TYPE DUT_HMI_General :
STRUCT
	Manuals 	: DUT_HMI_General_Manuals;		// Fanuc 
	Mes			: DUT_HMI_MesManual;
END_STRUCT
END_TYPE

(* stored: Version 1.1.0.1, ProductVersion 3.1.4024.15
   DUT DUT_HMI_General: Id {189f4ebb-88e4-4717-8022-bcfbb0cb8dc3} *)
